// TIA Portal V17 export
// export: Created 2022-02-03T14:45:10.2221615Z, ExportSetting WithDefaults, DisplayName Totally Integrated Automation Portal, DisplayVersion V17, DisplayName TIA Portal Openness, DisplayVersion V17, DisplayName TIA Portal Version Control Interface, DisplayVersion V17, DisplayName SINAMICS Startdrive Advanced, DisplayVersion V17, DisplayName SINAMICS Startdrive G130, G150, S120, S150, SINAMICS MV, S210, DisplayVersion V17, DisplayName SINAMICS Startdrive G110M, G120, G120C, G120D, G120P, G115D, DisplayVersion V17, DisplayName STEP 7 Professional, DisplayVersion V17, DisplayName STEP 7 Safety, DisplayVersion V17, DisplayName WinCC Advanced, DisplayVersion V17
ORGANIZATION_BLOCK "MainConveyor"   // OB1, LAD, ProgramCycle
TITLE = "Main Program Sweep (Cycle)"
VERSION : 0.1
// stored: AutoNumber true, IsIECCheckEnabled false, SetENOAutomatically false
   VAR_INPUT
      Initial_Call : Bool;   // Initial call of this OB
      Remanence : Bool;   // =True, if remanent data are available
   END_VAR
BEGIN

REGION Network 1
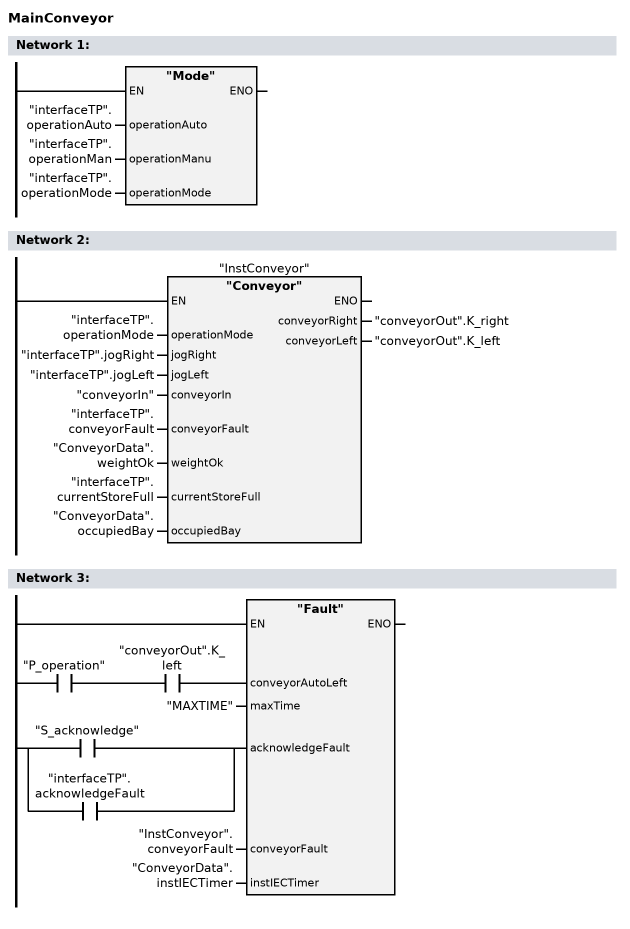
   RUNG wire#powerrail
      "Mode"(operationAuto := "interfaceTP".operationAuto, operationManu := "interfaceTP".operationMan, operationMode := "interfaceTP".operationMode)
   END_RUNG
   // the same network as SCL:
   "Mode"(operationAuto := "interfaceTP".operationAuto,
          operationManu := "interfaceTP".operationMan,
          operationMode := "interfaceTP".operationMode);
END_REGION

REGION Network 2
   RUNG wire#powerrail
      "InstConveyor"(operationMode := "interfaceTP".operationMode, jogRight := "interfaceTP".jogRight, jogLeft := "interfaceTP".jogLeft, conveyorIn := "conveyorIn", conveyorFault := "interfaceTP".conveyorFault, weightOk := "ConveyorData".weightOk, currentStoreFull := "interfaceTP".currentStoreFull, occupiedBay := "ConveyorData".occupiedBay, conveyorRight => "conveyorOut".K_right, conveyorLeft => "conveyorOut".K_left)
   END_RUNG
   // the same network as SCL:
   "InstConveyor"(operationMode := "interfaceTP".operationMode,   // "Conveyor"
                  jogRight := "interfaceTP".jogRight,
                  jogLeft := "interfaceTP".jogLeft,
                  conveyorIn := "conveyorIn",
                  conveyorFault := "interfaceTP".conveyorFault,
                  weightOk := "ConveyorData".weightOk,
                  currentStoreFull := "interfaceTP".currentStoreFull,
                  occupiedBay := "ConveyorData".occupiedBay,
                  conveyorRight => "conveyorOut".K_right,
                  conveyorLeft => "conveyorOut".K_left);
END_REGION

REGION Network 3
   RUNG wire#powerrail
      "Fault"(conveyorAutoLeft := wire#w1, acknowledgeFault := wire#w2, maxTime := "MAXTIME", conveyorFault := "InstConveyor".conveyorFault, instIECTimer := "ConveyorData".instIECTimer)
   END_RUNG
   RUNG wire#powerrail
      Contact( "P_operation" )
      Contact( "conveyorOut".K_left )
   END_RUNG wire#w1
   RUNG wire#powerrail
      Contact( "S_acknowledge" )
   END_RUNG wire#w2
   RUNG wire#powerrail
      Contact( "interfaceTP".acknowledgeFault )
   END_RUNG wire#w2
   // the same network as SCL:
   "Fault"(conveyorAutoLeft := "P_operation" AND "conveyorOut".K_left,
           maxTime := "MAXTIME",
           acknowledgeFault := "S_acknowledge" OR "interfaceTP".acknowledgeFault,
           conveyorFault := "InstConveyor".conveyorFault,
           instIECTimer := "ConveyorData".instIECTimer);
END_REGION
END_ORGANIZATION_BLOCK
